// TIA Portal V19 export
TYPE "LEXCHANGETRAY_typeConstraintWorkstation_toConstraintRollerDeliver"
// stored: Access Published
   STRUCT
      feedback : "LEXCHANGETRAY_typeConstraintWorkstationEm_toConstraintRollerFeedback";
      req : "LEXCHANGETRAY_typeConstraintWorkstationEm_toConstraintRollerReq";
   END_STRUCT;
END_TYPE
